TYPE ST180_Cylinders_e :
(
    Greifer_Patrone_Links,
    Greifer_Patrone_Rechts,
    Niederhalter_Deckel_Links,
    Niederhalter_Deckel_Rechts
);
END_TYPE

(* stored: Version 1.1.0.1, ProductVersion 3.1.4024.6
   EnumerationTextList ST180_Cylinders_e: Id {3cc58a29-6e17-4db7-9506-dcf36263dc61} *)
